FUNCTION_BLOCK Velocity_PI_LREAL2 (* Composite Function Block Type *)
  (* Standard: 61499-2 *)
  (* Version 0.0, 2018-07-28, 4DIAC-IDE, 4DIAC-Consortium *)
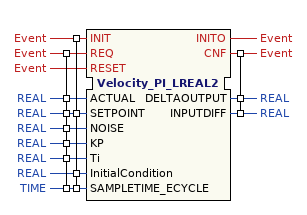
  EVENT_INPUT
    INIT WITH SAMPLETIME_ECYCLE, SETPOINT, InitialCondition; (* Initialization Request *)
    REQ WITH SAMPLETIME_ECYCLE, ACTUAL, SETPOINT, NOISE, KP, Ti; (* Normal Execution Request. disambung Event Cycle juga ya *)
    RESET;
  END_EVENT
  EVENT_OUTPUT
    INITO; (* Initialization Confirm *)
    CNF WITH DELTAOUTPUT, INPUTDIFF; (* Execution Confirmation *)
  END_EVENT
  VAR_INPUT
    ACTUAL : REAL;
    SETPOINT : REAL;
    NOISE : REAL;
    KP : REAL;
    Ti : REAL;
    InitialCondition : REAL;
    SAMPLETIME_ECYCLE : TIME;
  END_VAR
  VAR_OUTPUT
    DELTAOUTPUT : REAL;
    INPUTDIFF : REAL;
  END_VAR
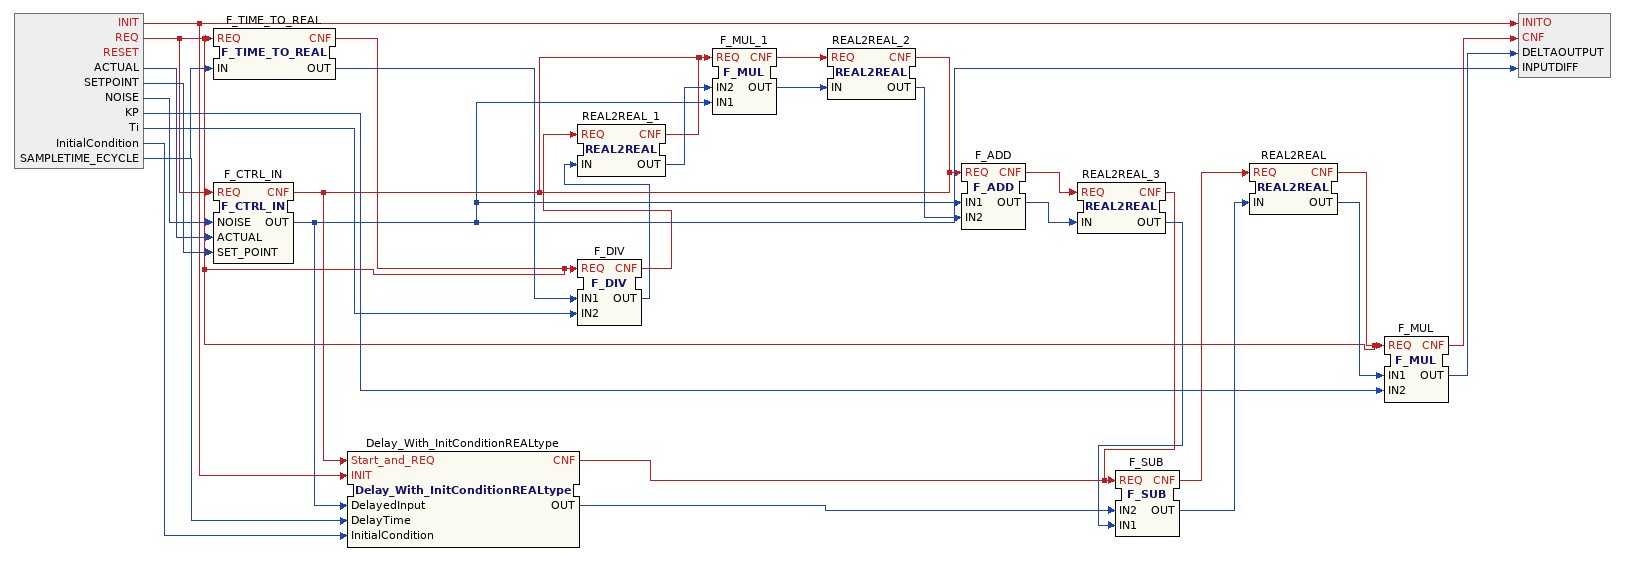
  FBS
    F_CTRL_IN : F_CTRL_IN;
    F_SUB : F_SUB;
    F_MUL : F_MUL;
    F_ADD : F_ADD;
    F_MUL_1 : F_MUL;
    F_DIV : F_DIV;
    REAL2REAL : REAL2REAL;
    F_TIME_TO_REAL : F_TIME_TO_REAL;
    Delay_With_InitConditionREALtype : Delay_With_InitConditionREALtype;
    REAL2REAL_1 : REAL2REAL;
    REAL2REAL_2 : REAL2REAL;
    REAL2REAL_3 : REAL2REAL;
  END_FBS
  EVENT_CONNECTIONS
    F_MUL.CNF TO CNF;
    F_SUB.CNF TO REAL2REAL.REQ;
    REAL2REAL.CNF TO F_MUL.REQ;
    REQ TO F_CTRL_IN.REQ;
    F_TIME_TO_REAL.CNF TO F_DIV.REQ;
    REQ TO F_DIV.REQ;
    REQ TO F_MUL.REQ;
    F_CTRL_IN.CNF TO Delay_With_InitConditionREALtype.Start_and_REQ;
    Delay_With_InitConditionREALtype.CNF TO F_SUB.REQ;
    F_DIV.CNF TO REAL2REAL_1.REQ;
    REAL2REAL_1.CNF TO F_MUL_1.REQ;
    F_CTRL_IN.CNF TO F_MUL_1.REQ;
    F_CTRL_IN.CNF TO F_ADD.REQ;
    REAL2REAL_2.CNF TO F_ADD.REQ;
    F_MUL_1.CNF TO REAL2REAL_2.REQ;
    REAL2REAL_3.CNF TO F_SUB.REQ;
    F_ADD.CNF TO REAL2REAL_3.REQ;
    INIT TO Delay_With_InitConditionREALtype.INIT;
    INIT TO INITO;
    REQ TO F_TIME_TO_REAL.REQ;
  END_CONNECTIONS
  DATA_CONNECTIONS
    F_SUB.OUT TO REAL2REAL.IN;
    REAL2REAL.OUT TO F_MUL.IN1;
    F_MUL.OUT TO DELTAOUTPUT;
    NOISE TO F_CTRL_IN.NOISE;
    ACTUAL TO F_CTRL_IN.ACTUAL;
    SETPOINT TO F_CTRL_IN.SET_POINT;
    SAMPLETIME_ECYCLE TO F_TIME_TO_REAL.IN;
    F_TIME_TO_REAL.OUT TO F_DIV.IN1;
    Ti TO F_DIV.IN2;
    KP TO F_MUL.IN2;
    F_CTRL_IN.OUT TO Delay_With_InitConditionREALtype.DelayedInput;
    SAMPLETIME_ECYCLE TO Delay_With_InitConditionREALtype.DelayTime;
    InitialCondition TO Delay_With_InitConditionREALtype.InitialCondition;
    Delay_With_InitConditionREALtype.OUT TO F_SUB.IN2;
    REAL2REAL_1.OUT TO F_MUL_1.IN2;
    F_DIV.OUT TO REAL2REAL_1.IN;
    F_CTRL_IN.OUT TO F_MUL_1.IN1;
    F_CTRL_IN.OUT TO INPUTDIFF;
    F_CTRL_IN.OUT TO F_ADD.IN1;
    F_MUL_1.OUT TO REAL2REAL_2.IN;
    REAL2REAL_2.OUT TO F_ADD.IN2;
    F_ADD.OUT TO REAL2REAL_3.IN;
    REAL2REAL_3.OUT TO F_SUB.IN1;
  END_CONNECTIONS
END_FUNCTION_BLOCK
